FUNCTION IsGoodData : BOOL// check into load data not nan and too big or too low
VAR_INPUT
	dataLr : LREAL;
END_VAR
VAR
END_VAR

IF LrealIsNaN( dataLr ) THEN
	IsGoodData := FALSE;
ELSIF dataLr > pmDev.InvalidValueEnergyIntoload OR dataLr <  0.0001 THEN
	IsGoodData := FALSE;
ELSE
	IsGoodData := True;
END_IF

END_FUNCTION

(* stored: Version 1.1.0.1, ProductVersion 3.1.4024.12
   POU IsGoodData: Id {980b0dff-4284-40d8-a89a-5ec6270dba4e}, SpecialFunc None *)
